FUNCTION_BLOCK FB_MotionAxisPowerNC IMPLEMENTS I_MotionAxisPower
VAR
END_VAR

END_FUNCTION_BLOCK

(* stored: Version 1.1.0.1
   POU FB_MotionAxisPowerNC: Id {2d321a15-46e6-4df8-9d45-5369c7f83c7c}, SpecialFunc None *)
